TYPE U_ARRAY_64 :
UNION
	
	WrnAryWord : ARRAY[0..3] OF WORD;
	WrnAryDWord : ARRAY[0..1] OF DWORD;
	WrnAryBit : ARRAY[0..63] OF BOOL;
	stTest: ST_WarningBits;
END_UNION
END_TYPE

(* stored: Version 1.1.0.1, ProductVersion 3.1.4026.18
   DUT U_ARRAY_64: Id {d4fd4ca8-af11-41a3-90af-92ffffb60385} *)
